RoboDK station: SistemaEnsamble.rdk

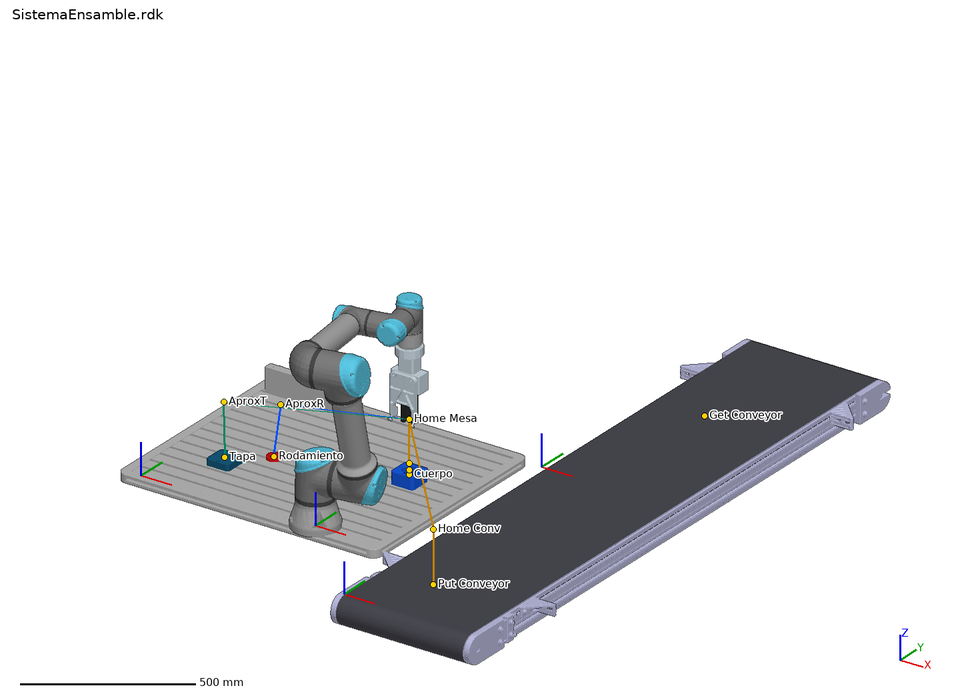
[picture v0: the station drawn from its stored meshes, robots at their saved joint values, targets as dots, program paths as lines]
Station SistemaEnsamble. Poses are relative to the parent item; angles as X-Y-Z fixed-axis rotations.
  - frame UR5e Base at (-323.09, 318.88, 0) mm
    - robot UR5e: 6 axes, payload 5 kg, reach 850 mm, repeatability 0.03 mm, weight 18.4 kg
        modified DH rows (alpha deg, a mm, theta deg, d mm): 0, 0, 0, 162.5; 90, 0, 180, 0; 0, 425, 0, 0; 0, 392.25, 0, 133.3; -90, 0, 0, 99.7; 90, 0, 180, 99.6
        joint limits [-360, -360, -360, -360, -360, -360] to [360, 360, 360, 360, 360, 360]; home [0, -90, -90, 0, 90, 0]; saved at [101.343, -72.239, -112.627, -85.134, 90, 11.343]
      - tool Gripper, TCP at (0, 0, 233.37) mm, size 100 x 89.2 x 240.5 mm
    - target Home Mesa (joint target) at (59.72, 380.06, 201) mm, rotated rx -180 ry 0 rz 0 deg; joints [101.343, -72.239, -112.627, -85.134, 90, 11.343] of UR5e
    - target Home Conv (joint target) at (524, -163.95, 201) mm, rotated rx 180 ry 0 rz 0 deg; joints [-3.323, -95.947, -91.559, -82.494, 90, -93.323] of UR5e
  - frame ConveyorReference at (0, 0, 0) mm
    - target Get Conveyor (Cartesian target) at (200, 1500, 20) mm, rotated rx 90 ry 0 rz -180 deg; joints [134.006, 22.86, -66.558, 43.699, -45.994, 0]
    - target Put Conveyor (Cartesian target) at (200.91, 154.93, 26) mm, rotated rx -180 ry 0 rz 0 deg; joints [-3.323, -104.313, -108.984, -56.703, 90, -93.323] of UR5e
    - object Conveyor at (0, 300, -50) mm, size 597 x 2090.8 x 107.2 mm
      - Python program RunConveyor (listed below)
      - Python program WaitForPart (listed below)
  - frame Mesa at (-13.37, 998.94, 0) mm
    - object Mesa at (0, 0, 0) mm, size 900 x 768.3 x 121 mm, geometry from Mesa.stl
  - frame Trabajo at (-913.37, 298.94, 1) mm
    - target Cuerpo (Cartesian target) at (650, 400, 25) mm, rotated rx -180 ry 0 rz 0 deg; joints [101.343, -81.79, -133.065, -55.144, 90, 11.343] of UR5e
    - target AproxR (Cartesian target) at (296.69, 268.66, 200.12) mm, rotated rx -179.98 ry 0 rz 58.66 deg; joints [160, -72.23, -112.62, -85.13, 90, 11.34] of UR5e
    - target Rodamiento (Cartesian target) at (250, 300, 10) mm, rotated rx -179.98 ry 0 rz 58.66 deg; joints [158.15, -91.704, -126.646, -51.63, 90.001, 9.49] of UR5e
    - target RodaCuer (Cartesian target) at (650, 400, 40) mm, rotated rx -180 ry 0 rz 0 deg; joints [101.343, -80.284, -131.642, -58.073, 90, 11.343] of UR5e
    - target AproxT (Cartesian target) at (155, 188.57, 200.26) mm, rotated rx -179.96 ry 0.01 rz 78.67 deg; joints [175.413, -84.405, -103.113, -82.443, 90.004, 6.743] of UR5e
    - target Tapa (Cartesian target) at (150.01, 200, 20) mm, rotated rx -179.96 ry 0.01 rz 78.67 deg; joints [174.028, -95.425, -120.781, -53.755, 90.005, 5.358] of UR5e
    - target Tapado (Cartesian target) at (650, 400.11, 60.1) mm, rotated rx -179.98 ry 0.01 rz -13.66 deg; joints [101.34, -78.5, -129.63, -61.85, 90, 25] of UR5e
    - object Part 3 T at (150, 200, 0) mm, size 80 x 80 x 20 mm, geometry from TAPA.stl
    - object Part 1 C at (650, 400, 0) mm, size 80 x 80 x 40 mm, geometry from Part1C.stl
    - object Part 2 R at (250, 300, 10) mm, size 45 x 45 x 11.5 mm, geometry from RODAMIENTO01.stl
  - program RESET (1 instructions, listed below)
  - program T_RODAMIENTO (7 instructions, listed below)
  - program P_RODAMIENTO (6 instructions, listed below)
  - program T_TAPA (7 instructions, listed below)
  - program P_TAPA (6 instructions, listed below)
  - program ENVIAR (15 instructions, listed below)
  - program MAIN (7 instructions, listed below)
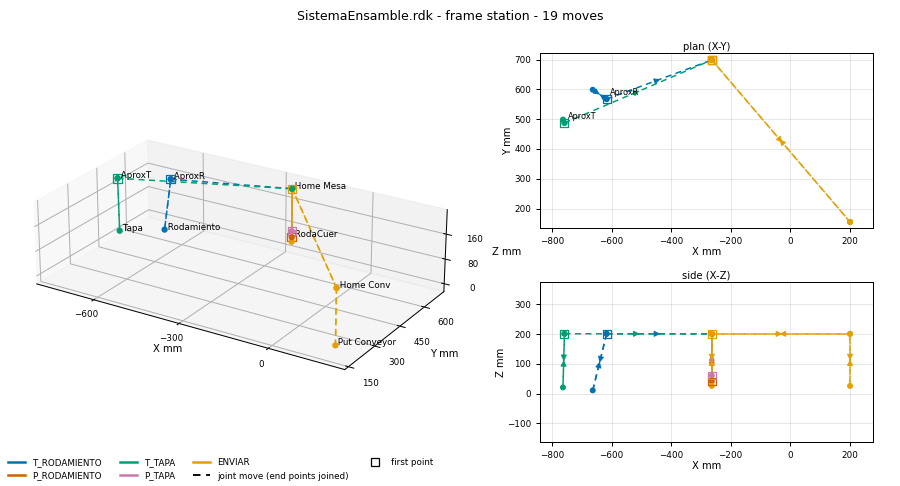
[picture p0: tool path of SistemaEnsamble.rdk in frame station, 19 of 19 moves have a stored position in this frame; points joined in program order, loops and branches not executed]

--- Python program RunConveyor ---
# Type help("robolink") or help("robodk") for more information
# Press F5 to run the script
# Note: you do not need to keep a copy of this file, your python script is saved with the station
from robolink import *    # API to communicate with RoboDK
from robodk import *      # basic matrix operations
RDK = Robolink()

# This script simulates a conveyor belt
CONVEYOR_NAME = 'Conveyor'
PICKABLE_OBJECTS_KEYWORD = 'Part'
# RDK.ShowMessage(CONVEYOR_NAME)
# Speed of movement in MM/S with respect to the conveyor coordinates:
MOVE_SPEED_MMS = [0,20,0]
REFRESH_RATE = 0.0050

# Define workspace of the conveyor to pick the objects:
CONV_SZ_X_MIN = 0
CONV_SZ_X_MAX = 440
CONV_SZ_Y_MIN = 0
CONV_SZ_Y_MAX = 2000
CONV_SZ_Z_MIN = -200
CONV_SZ_Z_MAX = +500

# Move objects that reached the end of the conveyor and were not picked:
FALLEN_OBJECTS = [0,0,-200]

# Get the conveyor item and reference for work space:
conv = RDK.Item(CONVEYOR_NAME)
conv_reference = conv.Parent()
poseconv = conv_reference.PoseAbs()

# One second in real life means 1 second of simulation. The simulation speed is taken from the station
SIMULATION_SPEED = 50

def is_inside_conveyor(pose):
    """Checks if a pose is inside the conveyor workspace"""
    pos = pose.Pos()
    if pos[0] > CONV_SZ_X_MIN and pos[0] < CONV_SZ_X_MAX and pos[1] > CONV_SZ_Y_MIN and pos[1] < CONV_SZ_Y_MAX and pos[2] > CONV_SZ_Z_MIN and pos[2] < CONV_SZ_Z_MAX:
        return True
    return False

def conveyor_move_object(pose, delta_time):
    """Moves the object pose through the conveyor depending on the time and speed"""
    delta_mm = mult3(MOVE_SPEED_MMS, delta_time)
    newpose = transl(delta_mm)*pose
    return newpose

# Get all objects (string list)
all_objects = RDK.ItemList(ITEM_TYPE_OBJECT, True)

# Convert object list into item pointers (faster)
# Also filter the list to take into account pickable objects only
objects = []
objects_name = []
objects_active = []
for i in range(len(all_objects)):
    if all_objects[i].count(PICKABLE_OBJECTS_KEYWORD) > 0:
        objects.append(RDK.Item(all_objects[i]))
        objects_name.append(all_objects[i])
        objects_active.append(False)

# The number of objects that can go in the conveyor
nobjects =len(objects)


# Infinite loop to simulate the conveyor behavior
current_time = 0
tic()
time_last = toc()
while True:
    # First: Look for objects that are not in the conveyor but are in the conveyor workspace
    for i in range(nobjects):
        obj_i = objects[i]

        # Skip if the object is already in the conveyor
        if objects_active[i]:
            continue

        # Check if the object has already been taken by a tool. If so, do not take it in the conveyor
        if obj_i.Parent().Type() == ITEM_TYPE_TOOL:
            continue

        # Check if the object is within the conveyor work area
        posei = obj_i.PoseAbs()
        poseirel = invH(poseconv)*posei
        if is_inside_conveyor(poseirel):
            # take the object
            obj_i.setParentStatic(conv)
            print('Objeto  %s colocado en el conveyor' % objects_name[i])
            objects_active[i] = True

    # Second step: Update the position of every object in the conveyor
    SIMULATION_SPEED = RDK.SimulationSpeed()
    time_current = toc()
    time_delta = time_current - time_last
    time_last = time_current
    current_time = current_time + time_delta*SIMULATION_SPEED

    # Make a list of objects with their matching positions to update
    obj_items = []
    obj_poses_abs = []
    for i in range(nobjects):
        obj_i = objects[i]

        # Check if the object has been picked from the conveyor
        if objects_active[i] and not obj_i.Parent().equals(conv):
            objects_active[i] = False
            print('Object %s was picked from the conveyor' % objects_name[i])
            continue

        # Skip update for objects that are not in the conveyor
        if not objects_active[i]:
            continue

        # Update the position of the object
        posei = invH(poseconv)*obj_i.PoseAbs()
        newposei = conveyor_move_object(posei, time_delta*SIMULATION_SPEED)
        if not is_inside_conveyor(newposei):
            print('Warning!! Object %s fell from the conveyor at %.1f seconds after simulation started' % (objects_name[i], current_time))
            #raise Exception('Object %s was not picked from the conveyor!' % objects_name[i])
            newposei = transl(FALLEN_OBJECTS)*newposei
            objects_active[i] = False

        #obj_i.setPose(newposei) # this will provoke a refresh (can be slow)
        obj_items.append(obj_i)
        obj_poses_abs.append(poseconv*newposei)

    # Update the object positions
    RDK.setPosesAbs(obj_items, obj_poses_abs)

    # Take a break...
    #pause(REFRESH_RATE)

--- Python program WaitForPart ---
# Type help("robolink") or help("robodk") for more information
# Press F5 to run the script
# Note: you do not need to keep a copy of this file, your python script is saved with the station
from robolink import *    # API to communicate with RoboDK
from robodk import *      # basic matrix operations
RDK = Robolink()

# This script allows to simulate a laser sensor
# that detect the presence of a part in a plane,
# such as a part crossing a laser sensor in a
# conveyor belt

# The script finishes once a part has been detected
# so it works like a WAIT UNTIL function.

# Use a target from the station as a reference plane:
TARGET_NAME = 'Get Conveyor'
LASER_PLANE = [0,-1,0] # normal of the plane

# Activate within this tolerance
TOLERANCE_CHECK_MM = 10

# Look for parts with the keyword "Part"
PICKABLE_OBJECTS_KEYWORD = 'Part'

# Update status every 1 ms
RECHECK_PERIOD = 0.001

# Get the target and the detection plane
target = RDK.Item(TARGET_NAME)
targetpose = target.PoseAbs()
DETECT_PLANE_POINT = targetpose.Pos()
DETECT_PLANE_VECTOR = LASER_PLANE

# Define a function to detect a target
def part_detected(pos):
    """Check if a part is in the detection area (proximity of a point to a plane)"""
    pos_proj = proj_pt_2_plane(pos, DETECT_PLANE_POINT, DETECT_PLANE_VECTOR)
    distance2plane = norm(subs3(pos,pos_proj))
    if distance2plane < TOLERANCE_CHECK_MM:
        return True
    return False

# Get all object names
all_objects = RDK.ItemList(ITEM_TYPE_OBJECT, True)

# Get object items in a list (faster) and filter by keyword
check_objects = []
check_objects_names = []
for i in range(len(all_objects)):
    if all_objects[i].count(PICKABLE_OBJECTS_KEYWORD) > 0:
        check_objects_names.append(all_objects[i])
        check_objects.append(RDK.Item(all_objects[i]))

# Make sure that there are part that we are expecting
nCheck_objects = len(check_objects)
if nCheck_objects == 0:
    raise Exception('No parts to check for. The keyword is %s.' % PICKABLE_OBJECTS_KEYWORD)

# Loop forever until a part is detected by the sensor
part_available = False;
while not part_available:
    for i in range(nCheck_objects):
        if part_detected(check_objects[i].PoseAbs().Pos()):
            print('Part detected: %s' % check_objects_names[i])
            part_available = True
            break

    # Wait some time...
    pause(RECHECK_PERIOD)

print('Procedure finished')

--- program RESET ---
  Reemplazar objetos

--- program T_RODAMIENTO (robot UR5e) ---
  Est. Ref.: Trabajo
  Est. herr: Gripper
  MoveJ (AproxR)
  MoveJ (Rodamiento)
  Adjuntar a Gripper
  MoveJ (AproxR)
  MoveJ (Home Mesa)

--- program P_RODAMIENTO (robot UR5e) ---
  Est. Ref.: Trabajo
  Est. herr: Gripper
  MoveJ (RodaCuer)
  Separar de Gripper
  Pausa 500 ms
  MoveJ (Home Mesa)

--- program T_TAPA (robot UR5e) ---
  Est. Ref.: Trabajo
  Est. herr: Gripper
  MoveJ (AproxT)
  MoveJ (Tapa)
  Adjuntar a Gripper
  MoveJ (AproxT)
  MoveJ (Home Mesa)

--- program P_TAPA (robot UR5e) ---
  Est. Ref.: Trabajo
  Est. herr: Gripper
  MoveJ (Tapado)
  Separar de Gripper
  MoveJ (Home Mesa)
  Pausa 1.5 s

--- program ENVIAR (robot UR5e) ---
  Est. Ref.: Trabajo
  Est. herr: Gripper
  MoveJ (Home Mesa)
  MoveJ (Target 1) -> target Cuerpo
  Adjuntar a Gripper
  Adjuntar a Gripper
  Adjuntar a Gripper
  MoveJ (Home Mesa)
  MoveJ (Home Conv)
  Est. Ref.: ConveyorReference
  MoveJ (Put Conveyor)
  Separar de Gripper
  Pausa 500 ms
  MoveJ (Home Conv)
  MoveJ (Home Mesa)

--- program MAIN (robot UR5e) ---
  Llamar RESET
  Ejecutar RunConveyor
  Llamar T_RODAMIENTO
  Llamar P_RODAMIENTO
  Llamar T_TAPA
  Llamar P_TAPA
  Llamar ENVIAR
